// TIA Portal V20 export
// export: Created 2025-12-01T14:57:20.2864517Z, ExportSetting None, DisplayName Totally Integrated Automation Portal, DisplayVersion V20 Update 3, DisplayName TIA Portal Openness, DisplayVersion V20 Update 3, DisplayName TIA Portal Version Control Interface, DisplayVersion V20 Update 3, DisplayName STEP 7 Professional, DisplayVersion V20 Update 3, DisplayName STEP 7 Safety, DisplayVersion V20 Update 2, DisplayName WinCC Basic/Comfort/Advanced, DisplayVersion V20 Update 3, DisplayName WinCC Professional, DisplayVersion V20 Update 3, DisplayName WinCC Unified, DisplayVersion V20 Update 3
DATA_BLOCK "DB230_CONTADORES"   // DB230
{ S7_Optimized_Access := 'FALSE' }
AUTHOR : ROUTER
// stored: AutoNumber false
   VAR
      Mesa : Array[0.."CTE_MaxMesas"] of Struct
         CNT_PRESENCIA : UDInt;
         CNT_AUSENCIA_ENTRADA : UDInt;
         CNT_AUSENCIA_SALIDA : UDInt;
         CNT_PARO : UDInt;
         CNT_Seg_HB_Avance : UDInt;
         CNT_Separacion_Sal : UDInt;
         CNT_Separacion_entrada : UDInt;
         CNT_CaraDelantera : UDInt;
         CNT_Reparto_E1 : UDInt;
         CNT_Reparto_E2 : UDInt;
         CNT_Reparto_E4 : UDInt;
         CNT_Detector_Fuera : UDInt;
         AUX_CNT : UDInt;
         CNT_Bloqueo_Movimiento : UDInt;
         CNT_Reposo : UDInt;
         CNT_Atasco : UDInt;
         CNT_Gap : UDInt;
         CNT_Acumulacion : UDInt;
         TMP_En_tension : UDInt;
         CNT_TopeE1S3 : UDInt;
         CNT_TopeE2S4 : UDInt;
         CNT_Transfer : UDInt;
         TMP_Decel_SM_E1S3 : UDInt;
         TMP_Decel_SM_E2S4 : UDInt;
         TMP_Decel_SM_ELEV : UDInt;
         MEM_OCUPACION : USInt;
      END_STRUCT;
   END_VAR
BEGIN
END_DATA_BLOCK
